Staubli VAL3: IO.pgx

program IO()
begin
end
